// TIA Portal project "MachineJob" (V18)

(* hardware
DEVICE "S7-1200 station_1"  S7-1200 Station
   slot 0: "Rack_0"  Rack  V1.0
   slot 1: "PLC_1"  CPU 1215C AC/DC/Rly  6ES7 215-1BG40-0XB0  V4.1
*)

// ===== PLC "PLC_1"  CPU 1215C AC/DC/Rly =====

VAR_GLOBAL   // PLC tag table "默认变量表"
   "MB_Server_NDR" AT %M10.1 : Bool;
   "MB_Server_DR" AT %M10.2 : Bool;
   "MB_Server_Error" AT %M10.3 : Bool;
   "MB_Server_Status" AT %MW100 : Word;
END_VAR

DATA_BLOCK "MachineJob_Data"   // DB1
{ S7_Optimized_Access := 'FALSE' }
VERSION : 0.1
   VAR
      Data1 : Word;
      Data2 : Word;
      Data3 : Word;
      Data4 : Word;
      Data5 : Word;
      Data6 : Word;
      Data7 : Word;
      Data8 : Word;
      Data9 : Word;
      Data10 : Word;
   END_VAR
BEGIN
END_DATA_BLOCK

DATA_BLOCK "MB_TCON"   // DB3
{ S7_Optimized_Access := 'FALSE' }
VERSION : 0.1
   VAR
      MB_Server : TCON_IP_v4;
   END_VAR
BEGIN
   MB_Server.InterfaceId := 64;
   MB_Server.ID := 2;
   MB_Server.LocalPort := 502;
END_DATA_BLOCK

ORGANIZATION_BLOCK "Main"   // OB1, LAD, ProgramCycle
TITLE = "Main Program Sweep (Cycle)"
{ S7_Optimized_Access := 'TRUE' }
VERSION : 0.1
   VAR_INPUT
      Initial_Call : Bool;   // Initial call of this OB
      Remanence : Bool;   // =True, if remanent data are available
   END_VAR
BEGIN

REGION Network 1
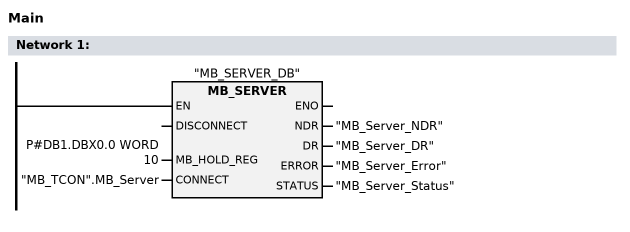
   "MB_SERVER_DB"(MB_HOLD_REG := P#DB1.DBX0.0 WORD 10,   // MB_SERVER
                  CONNECT := "MB_TCON".MB_Server,
                  NDR => "MB_Server_NDR",
                  DR => "MB_Server_DR",
                  ERROR => "MB_Server_Error",
                  STATUS => "MB_Server_Status");
END_REGION
END_ORGANIZATION_BLOCK